FUNCTION deltaReactivePwr_Voltage_Regulation : REAL
VAR_INPUT
	input: REAL;
END_VAR
VAR
	enhancedPoints: ARRAY [1..4, 1..3] OF REAL;
	 i: UINT;
	 x: REAL;
	 y: REAL;
	 g: REAL;
END_VAR

// 8.3.2.1. Regolazione della tensione ad anello aperto – Modalità Q(DV)
enhancedPoints[1][1] := -0.33;
enhancedPoints[1][2] := 0.1;
enhancedPoints[1][3] := -0.3125;

enhancedPoints[2][1] := -0.01;
enhancedPoints[2][2] := 0;
enhancedPoints[2][3] := 0;

enhancedPoints[3][1] := 0.01;
enhancedPoints[3][2] := 0;
enhancedPoints[3][3] := -0.3125;

enhancedPoints[4][1] := 0.33;
enhancedPoints[4][2] := -0.1;
enhancedPoints[4][3] := 0;


x := 0;
y := enhancedPoints[4][2];
g := 0;

IF (input <= enhancedPoints[1][1]) THEN
 	
	x := 0;
	y := enhancedPoints[1][2];
	g := 0;

ELSE 

	FOR i := 4 TO 1 BY -1 DO
		
		IF input < enhancedPoints[i][1] THEN
			CONTINUE;
		END_IF
		
		x := enhancedPoints[i][1];
		y := enhancedPoints[i][2];
		g := enhancedPoints[i][3];
		EXIT;
	
	END_FOR	

END_IF

deltaReactivePwr_Voltage_Regulation := y + g *(input - x);

END_FUNCTION

(* stored: Version 1.1.0.1, ProductVersion 3.1.4024.15
   POU deltaReactivePwr_Voltage_Regulation: Id {cff1b532-2074-4579-aaf1-e2b0151cd592}, SpecialFunc None *)
